(* Logix 5000 project; controller Prueba_Sintonizacion vendor 1 type 14 code 54 rev 20.11; software revision 20.00 *)

TASK MainTask (continuous, watchdog 500 ms) : MainProgram

MODULES
   Local : vendor 1 type 14 code 54 (ICP 0, rev 20.11)
END_MODULES

VAR_GLOBAL   (* controller tags *)
   Bit_prueba : BOOL;
   Caudal_1 : REAL;
   Caudal_2 : REAL;
   Caudal_Out_1 : REAL;
   Caudal_Out_2 : REAL;
   CV_TCV_201_1 : REAL;
   CV_TCV_202_1 : REAL;
   FI_Agua : REAL;
   FI_Vapor : REAL;
   Intercambiador_1 : BOOL;
   Intercambiador_2 : BOOL;
   PV_Temperature_1 : REAL;
   PV_Temperature_2 : REAL;
   T_Agua : REAL;
   T_Int_1 : REAL;
   T_Int_2 : REAL;
   T_vapor : REAL;
   TCV_201 : REAL;
   TCV_202 : REAL;
END_VAR

PROGRAM MainProgram   (* main routine MainRoutine *)
VAR
   PID : PID := (CTL := 8388608, PE := 1, SP := 30.0, KP := 0.029, KI := 61.247, KD := 15.352, MAXS := 100.0, MAXO := 100.0, UPD := 1.0, MAXI := 100.0, MAXCV := 100.0);
   PID2 : PID := (CTL := 41943040, CA := 1, PE := 1, SP := 60.0, KP := 0.013, KI := 71.98, KD := 17.99, MAXS := 100.0, MAXO := 100.0, UPD := 1.0, MAXI := 100.0, MAXCV := 100.0);
END_VAR

ROUTINE MainRoutine   (* ladder *)
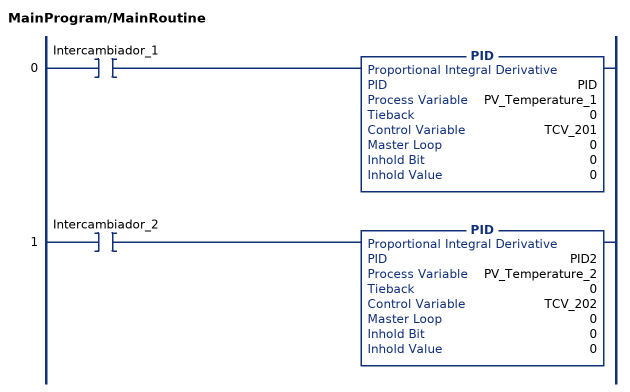
   0: XIC(Intercambiador_1)PID(PID,PV_Temperature_1,0,TCV_201,0,0,0);
   1: XIC(Intercambiador_2)PID(PID2,PV_Temperature_2,0,TCV_202,0,0,0);
END_ROUTINE
END_PROGRAM
